(* Logix 5000 project; controller Project1Template vendor 1 type 14 code 151 rev 33.12; software revision 33.01 *)

TASK MainTask (continuous, watchdog 500 ms) : MainProgram

MODULES
   Local : vendor 1 type 14 code 151 (Compact 0, rev 33.12)
      Discrete_IO : Embedded (Compact 1, rev 3.1, Output RPI 20 ms)
      Analog_IO : Embedded (Compact 2, rev 1.1, Output RPI 80 ms)
      Counters : Embedded (Compact 3, rev 1.1, Output RPI 20 ms)
END_MODULES

TYPE Part_Type :
STRUCT
   Part_Name : STRING;
   Part_Number : INT;
   F1_HL : REAL;
   F1_LL : REAL;
   F2_HL : REAL;
   F2_LL : REAL;
   F3_HL : REAL;
   F3_LL : REAL;
   F4_HL : REAL;
   F4_LL : REAL;
   Active : BOOL;
   F1_Count : COUNTER;
   F2_Count : COUNTER;
   F3_Count : COUNTER;
   F4_Count : COUNTER;
END_STRUCT
END_TYPE

TYPE SHIFT_DATA :
STRUCT
   COMPLETED : DINT;
   PASSED : DINT;
   FAILED : DINT;
   EFFICIENT : REAL;
END_STRUCT
END_TYPE

ADD_ON_INSTRUCTION AOI_SIM_2PosCyl_ExtRet   (* revision 1.0 *)
VAR_OUTPUT
   Animation : DINT; {visible}
END_VAR
VAR_INPUT
   TravelTime : DINT; {required}
   Extend_Output : BOOL; {required}
   Retract_Output : BOOL; {required}
END_VAR
VAR_OUTPUT
   Extend_Sensor : BOOL; {access Read Only, required}
   Retract_Sensor : BOOL; {access Read Only, required}
END_VAR
VAR_INPUT
   MCR : BOOL; {required}
   SingleSolenoidExtend : BOOL; {required}
   SingleSolenoidRetract : BOOL; {required}
   Retract_ValvePB : BOOL;
   Extend_ValvePB : BOOL;
END_VAR
VAR
   Extend_ScanCount : DINT;
   Retract_ScanCount : DINT; {access None}
   Extend_Timer : TIMER := (PRE := 500); {access None}
   Retract_Timer : TIMER := (PRE := 500); {access None}
   Retracted : BOOL; {access None}
   Extended : BOOL; {access None}
   Retract : BOOL; {access None}
   Extend : BOOL; {access None}
END_VAR

ROUTINE Logic   (* ladder *)
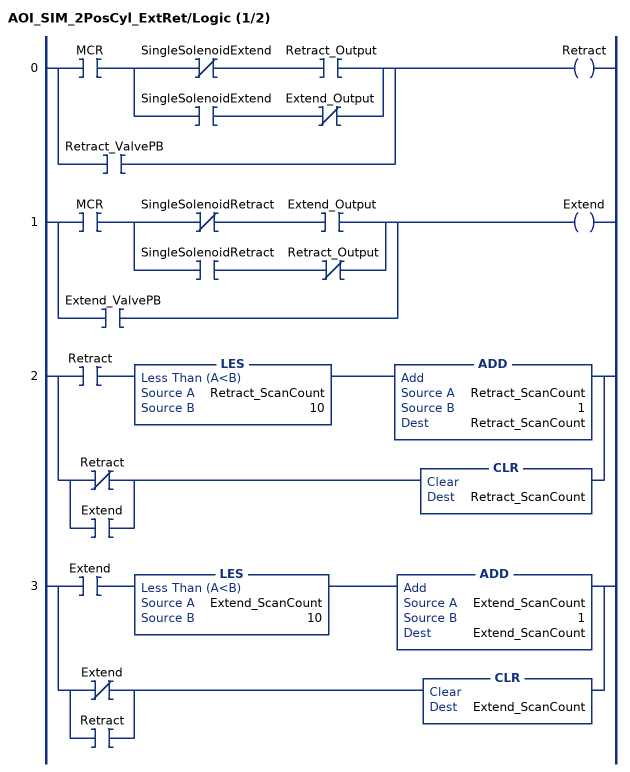
   0: [XIC(MCR) [XIO(SingleSolenoidExtend) XIC(Retract_Output) ,XIC(SingleSolenoidExtend) XIO(Extend_Output) ] ,XIC(Retract_ValvePB) ]OTE(Retract);
   1: [XIC(MCR) [XIO(SingleSolenoidRetract) XIC(Extend_Output) ,XIC(SingleSolenoidRetract) XIO(Retract_Output) ] ,XIC(Extend_ValvePB) ]OTE(Extend);
   2: [XIC(Retract) LES(Retract_ScanCount,10) ADD(Retract_ScanCount,1,Retract_ScanCount) ,[XIO(Retract) ,XIC(Extend) ] CLR(Retract_ScanCount) ];
   3: [XIC(Extend) LES(Extend_ScanCount,10) ADD(Extend_ScanCount,1,Extend_ScanCount) ,[XIO(Extend) ,XIC(Retract) ] CLR(Extend_ScanCount) ];
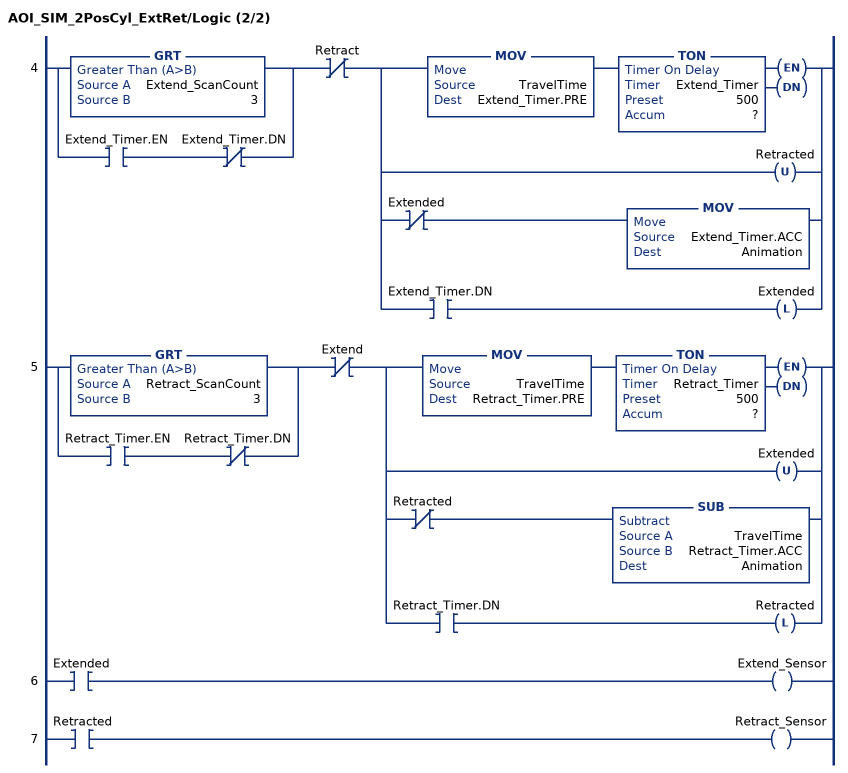
   4: [GRT(Extend_ScanCount,3) ,XIC(Extend_Timer.EN) XIO(Extend_Timer.DN) ]XIO(Retract)[MOV(TravelTime,Extend_Timer.PRE) TON(Extend_Timer,?,?) ,OTU(Retracted) ,XIO(Extended) MOV(Extend_Timer.ACC,Animation) ,XIC(Extend_Timer.DN) OTL(Extended) ];
   5: [GRT(Retract_ScanCount,3) ,XIC(Retract_Timer.EN) XIO(Retract_Timer.DN) ]XIO(Extend)[MOV(TravelTime,Retract_Timer.PRE) TON(Retract_Timer,?,?) ,OTU(Extended) ,XIO(Retracted) SUB(TravelTime,Retract_Timer.ACC,Animation) ,XIC(Retract_Timer.DN) OTL(Retracted) ];
   6: XIC(Extended)OTE(Extend_Sensor);
   7: XIC(Retracted)OTE(Retract_Sensor);
END_ROUTINE
END_ADD_ON_INSTRUCTION

ADD_ON_INSTRUCTION AOI_SIM_RandomDelay   (* revision 1.0 *)
VAR_INPUT
   Activate : BOOL; {access None}
   Target : DINT; {access None, required}
   Tolerance : DINT; {access None, required}
   PulseOutputTime : DINT; {access None, required}
END_VAR
VAR_OUTPUT
   DN : BOOL; {access Read Only, required}
END_VAR
VAR_INPUT
   DeActivate : BOOL; {access None}
END_VAR
VAR_OUTPUT
   TimingFirstHalf : BOOL; {access Read Only}
   TimingLastHalf : BOOL; {access Read Only}
   AccumlatedTime : DINT; {access Read Only}
   TT : BOOL; {access Read Only}
END_VAR
VAR
   StartTimerPulse : BOOL; {access None}
   StartTimerONS : BOOL; {access None}
   RandomIntermediate : DINT; {access None}
   RandomNumber : DINT; {access None}
   RandomPresetTime : DINT; {access None}
   RandomTimer : TIMER; {access None}
   PulseOutput : TIMER; {access None}
   Time50Percent : DINT; {access None}
END_VAR

ROUTINE Logic   (* ladder *)
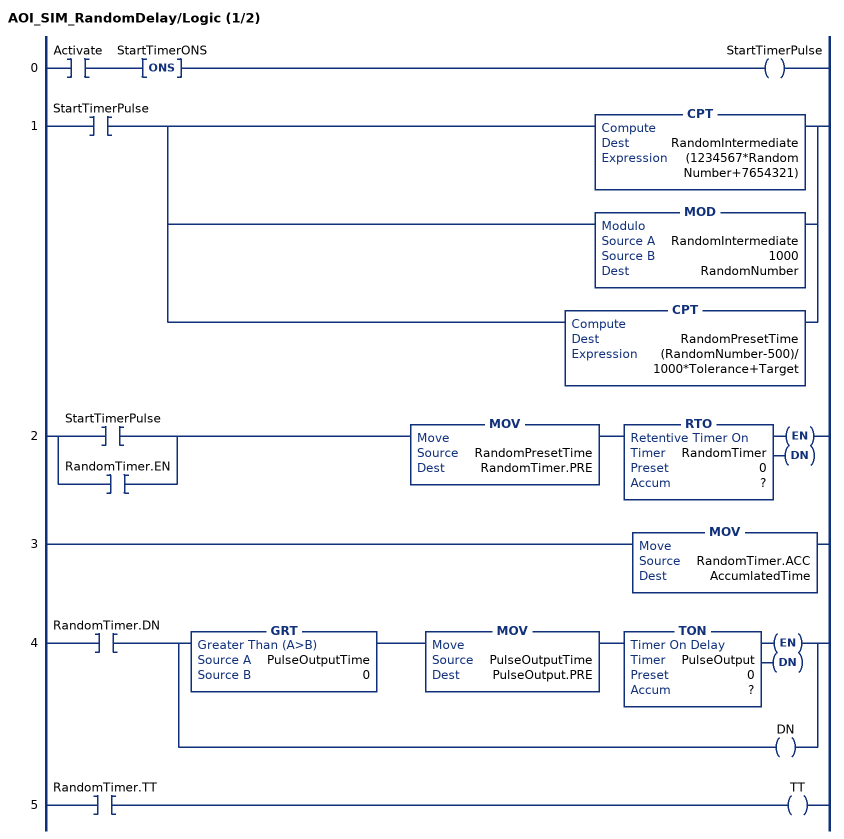
   0: XIC(Activate)ONS(StartTimerONS)OTE(StartTimerPulse);
   1: XIC(StartTimerPulse)[CPT(RandomIntermediate,(1234567*RandomNumber+7654321)) ,MOD(RandomIntermediate,1000,RandomNumber) ,CPT(RandomPresetTime,(RandomNumber-500)/1000*Tolerance+Target) ];
   2: [XIC(StartTimerPulse) ,XIC(RandomTimer.EN) ]MOV(RandomPresetTime,RandomTimer.PRE)RTO(RandomTimer,?,?);
   3: MOV(RandomTimer.ACC,AccumlatedTime);
   4: XIC(RandomTimer.DN)[GRT(PulseOutputTime,0) MOV(PulseOutputTime,PulseOutput.PRE) TON(PulseOutput,?,?) ,OTE(DN) ];
   5: XIC(RandomTimer.TT)OTE(TT);
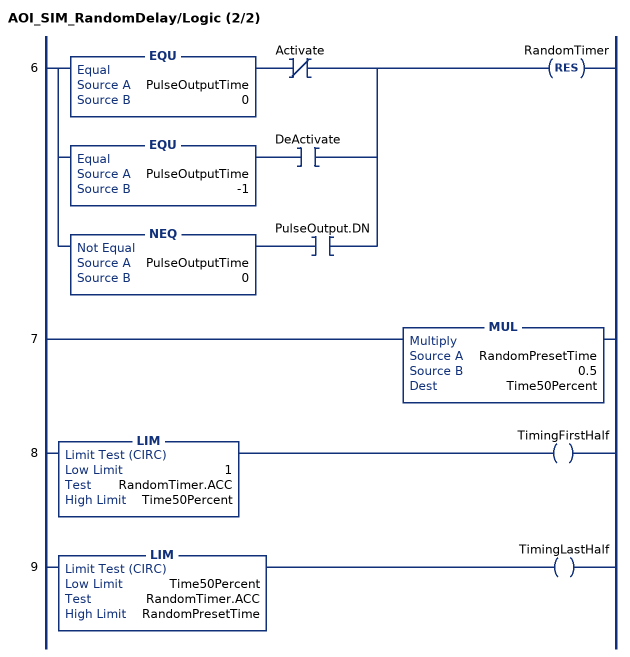
   6: [EQU(PulseOutputTime,0) XIO(Activate) ,EQU(PulseOutputTime,-1) XIC(DeActivate) ,NEQ(PulseOutputTime,0) XIC(PulseOutput.DN) ]RES(RandomTimer);
   7: MUL(RandomPresetTime,0.5,Time50Percent);
   8: LIM(1,RandomTimer.ACC,Time50Percent)OTE(TimingFirstHalf);
   9: LIM(Time50Percent,RandomTimer.ACC,RandomPresetTime)OTE(TimingLastHalf);
END_ROUTINE
END_ADD_ON_INSTRUCTION

ADD_ON_INSTRUCTION AOI_SIMAnalogSensor   (* revision 1.0 *)
VAR_IN_OUT
   Sensor : REAL; {required}
END_VAR
VAR_INPUT
   RampUpTime : DINT; {required}
   RampDwnTime : DINT; {required}
   Min : REAL; {required}
   Max : REAL; {required}
   Target : REAL; {required}
   Tolerance : REAL; {required}
   Fluctuation : REAL; {access None, required}
   Activate : BOOL; {access None}
END_VAR
VAR
   RampUpTimer : TIMER; {access None}
   RampDwnTimer : TIMER; {access None}
   FluctuateTimer : TIMER; {access None}
   FluctuateONS : BOOL; {access None}
   CurrentValue : REAL; {access Read Only}
   RampDwnTriggerONS : BOOL; {access Read Only}
   RampDwnTriggerPulse : BOOL; {access Read Only}
   RampUpTriggerONS : BOOL; {access Read Only}
   RampUpTriggerPulse : BOOL; {access Read Only}
   RandomNumber : DINT; {access Read Only}
   RandomTarget : REAL; {access Read Only}
   RandomIntermediate : DINT; {access Read Only}
   ScaledRampDwnTime : REAL; {access Read Only}
   ScaledRampUpTime : REAL; {access Read Only}
   Fluctuate : BOOL; {access None}
END_VAR

ROUTINE Logic   (* ladder *)
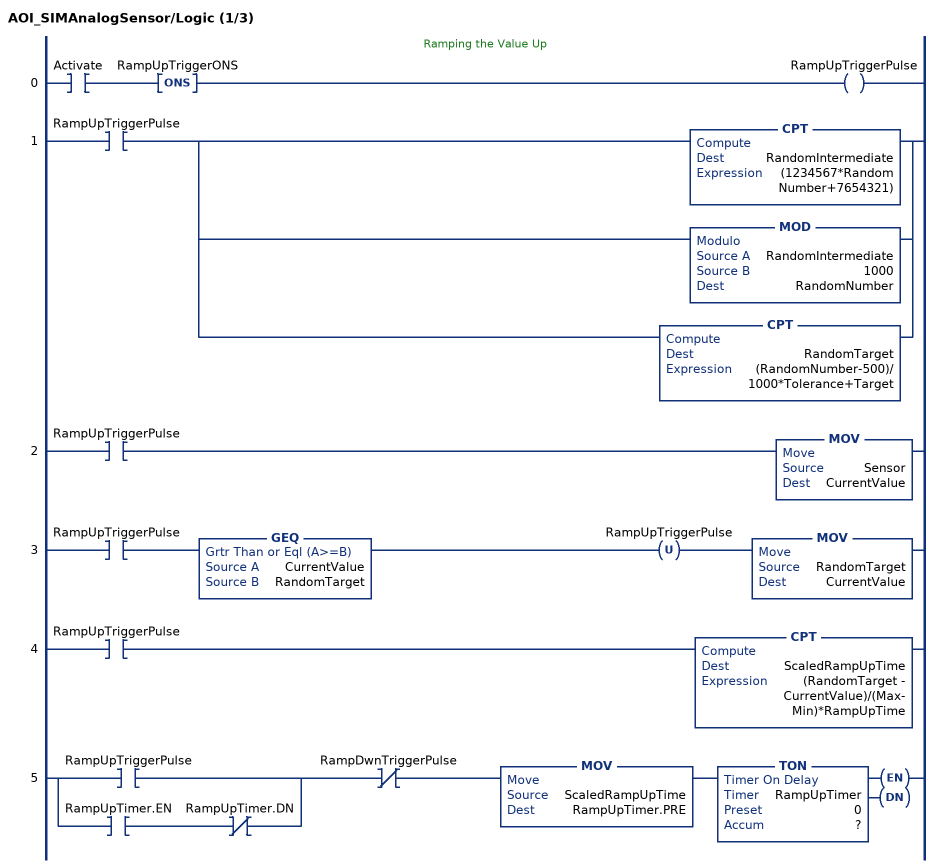
   // Ramping the Value Up
   0: XIC(Activate)ONS(RampUpTriggerONS)OTE(RampUpTriggerPulse);
   1: XIC(RampUpTriggerPulse)[CPT(RandomIntermediate,(1234567*RandomNumber+7654321)) ,MOD(RandomIntermediate,1000,RandomNumber) ,CPT(RandomTarget,(RandomNumber-500)/1000*Tolerance+Target) ];
   2: XIC(RampUpTriggerPulse)MOV(Sensor,CurrentValue);
   3: XIC(RampUpTriggerPulse)GEQ(CurrentValue,RandomTarget)OTU(RampUpTriggerPulse)MOV(RandomTarget,CurrentValue);
   4: XIC(RampUpTriggerPulse)CPT(ScaledRampUpTime,(RandomTarget - CurrentValue)/(Max-Min)*RampUpTime);
   5: [XIC(RampUpTriggerPulse) ,XIC(RampUpTimer.EN) XIO(RampUpTimer.DN) ]XIO(RampDwnTriggerPulse)MOV(ScaledRampUpTime,RampUpTimer.PRE)TON(RampUpTimer,?,?);
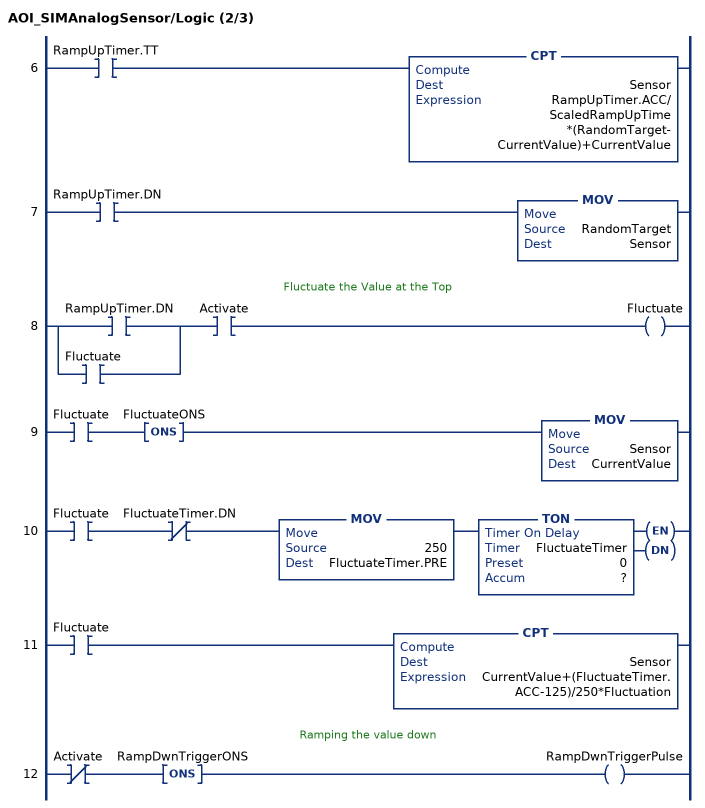
   6: XIC(RampUpTimer.TT)CPT(Sensor,RampUpTimer.ACC/ScaledRampUpTime *(RandomTarget-CurrentValue)+CurrentValue);
   7: XIC(RampUpTimer.DN)MOV(RandomTarget,Sensor);
   // Fluctuate the Value at the Top
   8: [XIC(RampUpTimer.DN) ,XIC(Fluctuate) ]XIC(Activate)OTE(Fluctuate);
   9: XIC(Fluctuate)ONS(FluctuateONS)MOV(Sensor,CurrentValue);
   10: XIC(Fluctuate)XIO(FluctuateTimer.DN)MOV(250,FluctuateTimer.PRE)TON(FluctuateTimer,?,?);
   11: XIC(Fluctuate)CPT(Sensor,CurrentValue+(FluctuateTimer.ACC-125)/250*Fluctuation);
   // Ramping the value down
   12: XIO(Activate)ONS(RampDwnTriggerONS)OTE(RampDwnTriggerPulse);
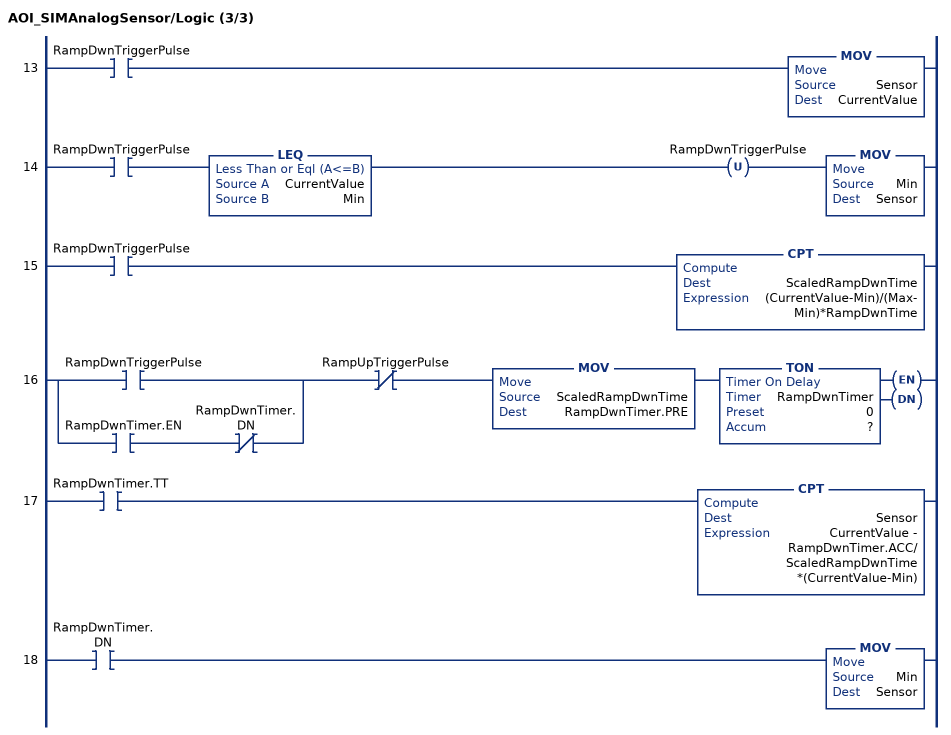
   13: XIC(RampDwnTriggerPulse)MOV(Sensor,CurrentValue);
   14: XIC(RampDwnTriggerPulse)LEQ(CurrentValue,Min)OTU(RampDwnTriggerPulse)MOV(Min,Sensor);
   15: XIC(RampDwnTriggerPulse)CPT(ScaledRampDwnTime,(CurrentValue-Min)/(Max-Min)*RampDwnTime);
   16: [XIC(RampDwnTriggerPulse) ,XIC(RampDwnTimer.EN) XIO(RampDwnTimer.DN) ]XIO(RampUpTriggerPulse)MOV(ScaledRampDwnTime,RampDwnTimer.PRE)TON(RampDwnTimer,?,?);
   17: XIC(RampDwnTimer.TT)CPT(Sensor,CurrentValue - RampDwnTimer.ACC/ScaledRampDwnTime *(CurrentValue-Min));
   18: XIC(RampDwnTimer.DN)MOV(Min,Sensor);
END_ROUTINE
END_ADD_ON_INSTRUCTION

VAR_GLOBAL   (* controller tags *)
   A_EXT_TMR : TIMER := (PRE := 10000);
   A_RET_TMR : TIMER := (PRE := 10000);
   ADD12 : DINT := 4;
   ADD123 : DINT := 6;
   ADD123FAIL : DINT := 3;
   ADD123PASS : DINT := 3;
   ADD12FAIL : DINT := 2;
   ADD12PASS : DINT := 2;
   ALLFAILONES : BOOL;
   AVERAGE1 : CONTROL := (LEN := 50);
   AVERAGECNTRL : CONTROL := (LEN := 50);
   B_EXT_TMR : TIMER := (PRE := 10000);
   B_RET_TMR : TIMER := (PRE := 10000);
   Batch_Count : INT;
   C_EXT_TMR : TIMER := (PRE := 10000);
   C_RET_TMR : TIMER := (PRE := 10000);
   CHANGED : BOOL;
   CHANGEONS : BOOL;
   Current_Part : Part_Type;
   Current_Part_Count : INT;
   Current_Part_Name : STRING;
   Current_Part_Number : INT;
   CURRENT_SHIFT : SHIFT_DATA := (COMPLETED := 8, PASSED := 5, FAILED := 3, EFFICIENT := 62.5);
   CURRENT_TOTAL_COUNT : DINT;
   DATASHIFT : BOOL;
   EFFICIENCY : REAL;
   END_SHIFT_PB : BOOL;
   EStop : BOOL;
   EXTRA_TIME : TIMER := (PRE := 120000);
   F1_AVERAGE : REAL := 44.42104;
   F1_Count : COUNTER := (ACC := 2, DN := 1);
   F1_CT_AVERAGE : REAL := 1000.2;
   F1_CT_History : REAL[5] := ([0] := 2501.0, [2] := 2500.0);
   F1_Current_Part_Count : DINT;
   F1_FAIL : COUNTER := (ACC := 1, DN := 1);
   F1_PASS : COUNTER := (ACC := 1, DN := 1);
   F1_TEMP_TORQUE : DINT[50];
   F1_TORQUE : REAL[50];
   F1_Torque_History : REAL[5] := ([0] := 75.627594, [1] := 73.2388, [2] := 73.2388);
   F2_Count : COUNTER := (ACC := 2, DN := 1);
   F2_CT_AVERAGE : REAL := 3399.4;
   F2_CT_History : REAL[5] := ([0] := 3499.0, [2] := 13498.0);
   F2_Current_Part_Count : DINT;
   F2_FAIL : COUNTER := (ACC := 1, DN := 1);
   F2_PASS : COUNTER := (ACC := 1, DN := 1);
   F2_Torque_History : REAL[5] := ([0] := 74.103195, [1] := 73.3064, [2] := 73.3064);
   F3_Count : COUNTER := (ACC := 2, DN := 1);
   F3_CT_AVERAGE : REAL := 3799.8;
   F3_CT_History : REAL[5] := ([0] := 4499.0, [2] := 14500.0);
   F3_Current_Part_Count : DINT;
   F3_FAIL : COUNTER := (ACC := 1, DN := 1);
   F3_PASS : COUNTER := (ACC := 1, DN := 1);
   F3_Torque_History : REAL[5] := ([0] := 76.578, [1] := 72.995605, [2] := 72.995605);
   F4_Count : COUNTER := (ACC := 2, DN := 1);
   F4_CT_AVERAGE : REAL := 3499.6;
   F4_CT_History : REAL[5] := ([0] := 3749.0, [2] := 13749.0);
   F4_Current_Part_Count : DINT;
   F4_FAIL : COUNTER := (DN := 1);
   F4_PASS : COUNTER := (ACC := 2, DN := 1);
   F4_Torque_History : REAL[5] := ([0] := 78.5, [1] := 77.1048, [2] := 77.1048);
   F_ALL_CTR : COUNTER := (ACC := 1);
   FAILONS1 : BOOL;
   FAILONS2 : BOOL;
   FAILONS3 : BOOL;
   FAILONS4 : BOOL;
   FASTEN_AllComplete : BOOL;
   FASTEN_AllTorquesFail : BOOL;
   FASTEN_AllTorquesPass : BOOL;
   FASTEN_F1Complete : BOOL;
   FASTEN_F1Complete_ONS : BOOL;
   FASTEN_F1Torque : REAL;
   FASTEN_F1TorqueFail : BOOL;
   FASTEN_F1TorquePass : BOOL;
   FASTEN_F2Complete : BOOL;
   FASTEN_F2Complete_ONS : BOOL;
   FASTEN_F2Torque : REAL;
   FASTEN_F2TorqueFail : BOOL;
   FASTEN_F2TorquePass : BOOL;
   FASTEN_F3Complete : BOOL;
   FASTEN_F3Complete_ONS : BOOL;
   FASTEN_F3Torque : REAL;
   FASTEN_F3TorqueFail : BOOL;
   FASTEN_F3TorquePass : BOOL;
   FASTEN_F4Complete : BOOL;
   FASTEN_F4Complete_ONS : BOOL;
   FASTEN_F4Torque : REAL;
   FASTEN_F4TorqueFail : BOOL;
   FASTEN_F4TorquePass : BOOL;
   FASTEN_TorqueFeedback : REAL := 20.050001;
   FAULTRESET_PB : BOOL;
   FAULTS : DINT;
   FAULTSIND : BOOL;
   FIX_EXT_TMR : TIMER := (PRE := 10000);
   FIX_RET_TMR : TIMER := (PRE := 10000);
   FIXTURE_AllPartsPresent : BOOL := 1;
   FIXTURE_AtHomePos : BOOL := 1;
   FIXTURE_Empty : BOOL;
   FIXTURE_PartsSecured : BOOL;
   FIXTURE_PartsSecuredTmr : TIMER := (PRE := 500);
   FromHMI_ExtClampA_PB : BOOL;
   FromHMI_ExtClampB_PB : BOOL;
   FromHMI_ExtClampC_PB : BOOL;
   FromHMI_ExtFixture_PB : BOOL;
   FromHMI_F1LowLim : REAL := 50.0;
   FromHMI_F1UppLim : REAL := 95.0;
   FromHMI_F2LowLim : REAL := 65.0;
   FromHMI_F2UppLim : REAL := 85.0;
   FromHMI_F3LowLim : REAL := 60.0;
   FromHMI_F3UppLim : REAL := 85.0;
   FromHMI_F4LowLim : REAL := 66.0;
   FromHMI_F4UppLim : REAL := 95.0;
   FromHMI_RetClampA_PB : BOOL;
   FromHMI_RetClampB_PB : BOOL;
   FromHMI_RetClampC_PB : BOOL;
   FromHMI_RetFixture_PB : BOOL;
   FROMHMI_SCREEN : DINT;
   FromHMI_StartPB : BOOL;
   FromHMI_StopPB : BOOL;
   FromRbt_ClearOfFixture : BOOL := 1;
   FromRbt_Fasten1Complete : BOOL;
   FromRbt_Fasten2Complete : BOOL;
   FromRbt_Fasten3Complete : BOOL;
   FromRbt_Fasten4Complete : BOOL;
   HomePB : BOOL;
   Honda : STRING := 'Honda';
   I1 : INT := 20318;
        .10   // Part Present C Sensor
        .11   // Part Present D Sensor
        .14   // Light Curtain Safety Circuit
        .0   // Fixture at Robot Limit Switch
        .1   // Fixture at Operator Limit Switch
        .2   // Clamp A Retracted Limit Switch
        .3   // Clamp B Retracted Limit Switch
        .4   // Clamp C Retracted Limit Switch
        .8   // Part Present A Sensor
        .9   // Part Present B Sensor
   I2_CHA : REAL := 4.01;   // Torque Sensor Input
   Lexus : STRING := 'Lexus';
   Load_PB : BOOL;
   O3 : INT;
        .1   // Fixture Retract to Operator
        .3   // Clamp B Extend Solenoid
        .0   // Fixture Extend to Robot
        .2   // Clamp A Extend Solenoid
        .4   // Clamp C Extend Solenoid
   ONEHR : BOOL;
   ONS1 : BOOL;
   ONS2 : BOOL;
   ONS3 : BOOL;
   ONS4 : BOOL;
   P1_ADD12 : DINT;
   P1_ADD123 : DINT;
   P2_ADD12 : DINT;
   P2_ADD123 : DINT;
   P3_ADD12 : DINT;
   P3_ADD123 : DINT;
   PART1 : Part_Type := (Part_Name := 'toyota', Part_Number := 1, F1_HL := 95.0, F1_LL := 75.0, F2_HL := 85.0, F2_LL := 75.0, F3_HL := 85.0, F3_LL := 75.0, F4_HL := 95.0, F4_LL := 75.0, F1_Count.DN := 1, F2_Count.DN := 1, F3_Count.DN := 1, F4_Count.DN := 1);
   PART2 : Part_Type := (F1_Count.DN := 1, F2_Count.DN := 1, F3_Count.DN := 1, F4_Count.DN := 1);
   PART3 : Part_Type := (Part_Name := 'Honda', Part_Number := 3, F1_HL := 95.0, F1_LL := 50.0, F2_HL := 85.0, F2_LL := 65.0, F3_HL := 85.0, F3_LL := 60.0, F4_HL := 95.0, F4_LL := 66.0, F1_Count.DN := 1, F2_Count.DN := 1, F3_Count.DN := 1, F4_Count.DN := 1);
   Part_Name : STRING;
   Part_Number : DINT := 3;
   Requested_Part_Number : INT;
   RESET_STATS : BOOL;
   S1ON : BOOL;
   SCREENREQTMR : TIMER := (PRE := 1000);
   SHIFT1ONS : BOOL;
   SHIFT_CHANGE : BOOL;
   SHIFT_TIMER : TIMER := (PRE := 120000);
   SHIFTHISTORY : SHIFT_DATA[5];
   SHIFTONS : BOOL;
   STARTONS : BOOL;
   SYS_AutoModeActive : BOOL := 1;
   SYS_CycleActive : BOOL;
   SYS_ManualModeActive : BOOL;
   SYS_StartPBPulseTmr : TIMER := (PRE := 200);
   T1AVG : DINT;
   THREEHR : BOOL;
   TIME : REAL;
   TOHMI_CHANGEVALVE : BOOL;
   TOHMI_CHANGEWARNING : BOOL;
   TOHMI_SCREENREQ : DINT;
   ToRbt_Fasten1Start : BOOL;
   ToRbt_Fasten2Start : BOOL;
   ToRbt_Fasten3Start : BOOL;
   ToRbt_Fasten4Start : BOOL;
   Total_Parts : INT;
   TOTAL_PARTS_COMPLETE : DINT;
   TOTAL_PARTS_FAIL : DINT;
   TOTAL_PARTS_PASS : DINT;
   Toyota : STRING := 'toyota';
   TWOHR : BOOL;
   VALVECTR : COUNTER := (ACC := 10, DN := 1);
   VALVEONS : BOOL;
   VALVEWARNING : DINT;
END_VAR

PROGRAM MainProgram   (* main routine MainRoutine *)
VAR
   Cycle_Time_Calc : TIMER := (PRE := 9999999);
   F1_CycleTime : REAL := 2501.0;
   F2_AVERAGE : REAL := 44.143196;
   F2_CycleTime : REAL := 3499.0;
   F2_TMR : TIMER := (PRE := 9999999);
   F3_AVERAGE : REAL := 44.513844;
   F3_CycleTime : REAL := 4499.0;
   F3_TMR : TIMER := (PRE := 9999999);
   F4_AVERAGE : REAL := 46.54192;
   F4_CycleTime : REAL := 3749.0;
   F4_TMR : TIMER := (PRE := 9999999);
   ONS_CTH : BOOL;
   ONS_F1_CT : BOOL;
   ONS_TH : BOOL;
   SIM_ClampA : AOI_SIM_2PosCyl_ExtRet := (TravelTime := 1000, Retract_Sensor := 1, MCR := 1, SingleSolenoidExtend := 1);
   SIM_ClampB : AOI_SIM_2PosCyl_ExtRet := (TravelTime := 1250, Retract_Sensor := 1, MCR := 1, SingleSolenoidExtend := 1);
   SIM_ClampC : AOI_SIM_2PosCyl_ExtRet := (TravelTime := 1250, Retract_Sensor := 1, MCR := 1, SingleSolenoidExtend := 1);
   SIM_EmptyFixture : TIMER := (PRE := 15000);
   SIM_Fasten1 : AOI_SIM_RandomDelay := (Target := 2500, Tolerance := 750);
   SIM_Fasten2 : AOI_SIM_RandomDelay := (Target := 3500, Tolerance := 450);
   SIM_Fasten3 : AOI_SIM_RandomDelay := (Target := 4500, Tolerance := 250);
   SIM_Fasten4 : AOI_SIM_RandomDelay := (Target := 3750, Tolerance := 500);
   SIM_Fixture : AOI_SIM_2PosCyl_ExtRet := (TravelTime := 2000, Retract_Sensor := 1, MCR := 1);
   SIM_LightCurtainPartPlace : AOI_SIM_RandomDelay := (Target := 6000, Tolerance := 1500, PulseOutputTime := 50);
   SIM_LightCurtainPartRem : AOI_SIM_RandomDelay := (Target := 5000, Tolerance := 1000, PulseOutputTime := 50);
   SIM_NOP : BOOL;
   SIM_Oneshots : DINT := 1;
   SIM_OperatorWorking : AOI_SIM_RandomDelay := (Target := 4000, Tolerance := 2000, PulseOutputTime := 50);
   SIM_PP_OFF : AOI_SIM_RandomDelay := (Target := 2500, Tolerance := 1000, PulseOutputTime := 50);
   SIM_PPA_ON : AOI_SIM_RandomDelay := (Target := 1500, Tolerance := 500, PulseOutputTime := 50);
   SIM_PPB_ON : AOI_SIM_RandomDelay := (Target := 2000, Tolerance := 1000, PulseOutputTime := 50);
   SIM_PPC_ON : AOI_SIM_RandomDelay := (Target := 2500, Tolerance := 1000, PulseOutputTime := 50);
   SIM_PPD_ON : AOI_SIM_RandomDelay := (Target := 3000, Tolerance := 500, PulseOutputTime := 50);
   SIM_RobotClear : AOI_SIM_RandomDelay := (Target := 1200, Tolerance := 250, PulseOutputTime := 50);
   SIM_Torque : AOI_SIMAnalogSensor := (RampUpTime := 500, RampDwnTime := 50, Min := 4.01, Max := 19.99, Target := 15.0, Tolerance := 2.0, Fluctuation := 0.04);
END_VAR

ROUTINE EXTRAS   (* ladder *)
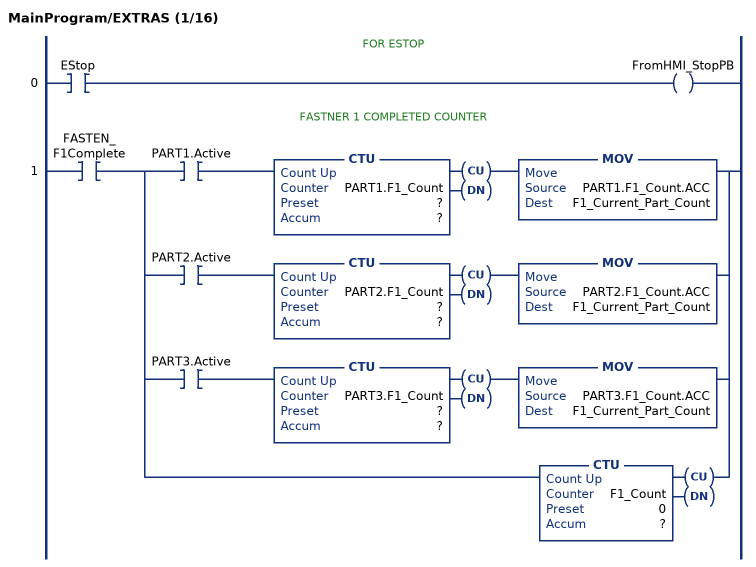
   // FOR ESTOP
   0: XIC(EStop)OTE(FromHMI_StopPB);
   // FASTNER 1 COMPLETED COUNTER
   1: XIC(FASTEN_F1Complete)[XIC(PART1.Active) CTU(PART1.F1_Count,?,?) MOV(PART1.F1_Count.ACC,F1_Current_Part_Count) ,XIC(PART2.Active) CTU(PART2.F1_Count,?,?) MOV(PART2.F1_Count.ACC,F1_Current_Part_Count) ,XIC(PART3.Active) CTU(PART3.F1_Count,?,?) MOV(PART3.F1_Count.ACC,F1_Current_Part_Count) ,CTU(F1_Count,?,?) ];
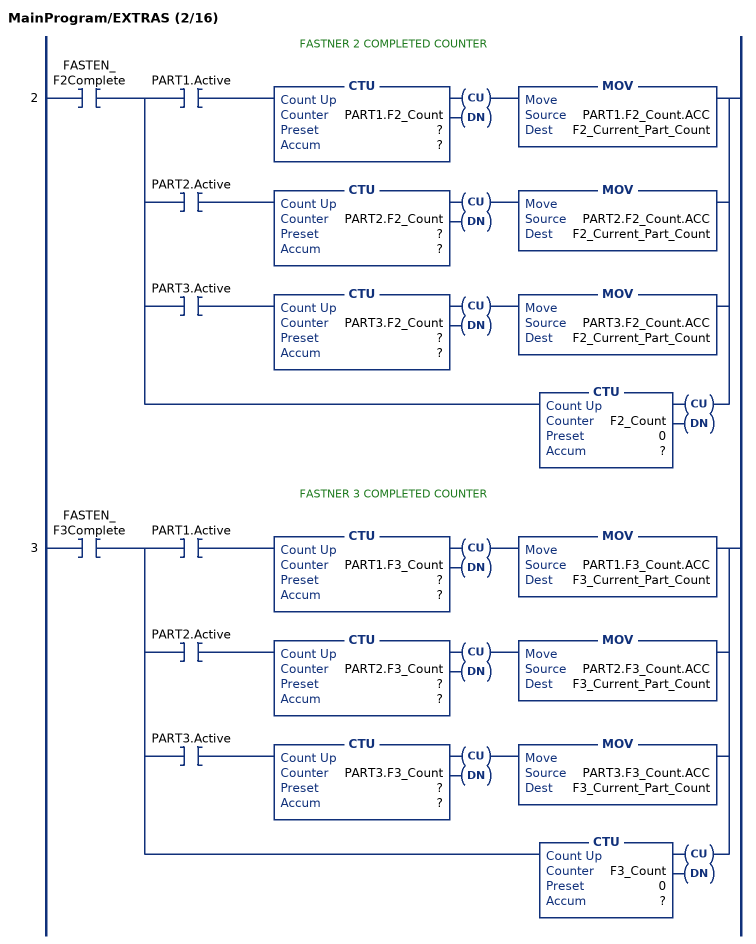
   // FASTNER 2 COMPLETED COUNTER
   2: XIC(FASTEN_F2Complete)[XIC(PART1.Active) CTU(PART1.F2_Count,?,?) MOV(PART1.F2_Count.ACC,F2_Current_Part_Count) ,XIC(PART2.Active) CTU(PART2.F2_Count,?,?) MOV(PART2.F2_Count.ACC,F2_Current_Part_Count) ,XIC(PART3.Active) CTU(PART3.F2_Count,?,?) MOV(PART3.F2_Count.ACC,F2_Current_Part_Count) ,CTU(F2_Count,?,?) ];
   // FASTNER 3 COMPLETED COUNTER
   3: XIC(FASTEN_F3Complete)[XIC(PART1.Active) CTU(PART1.F3_Count,?,?) MOV(PART1.F3_Count.ACC,F3_Current_Part_Count) ,XIC(PART2.Active) CTU(PART2.F3_Count,?,?) MOV(PART2.F3_Count.ACC,F3_Current_Part_Count) ,XIC(PART3.Active) CTU(PART3.F3_Count,?,?) MOV(PART3.F3_Count.ACC,F3_Current_Part_Count) ,CTU(F3_Count,?,?) ];
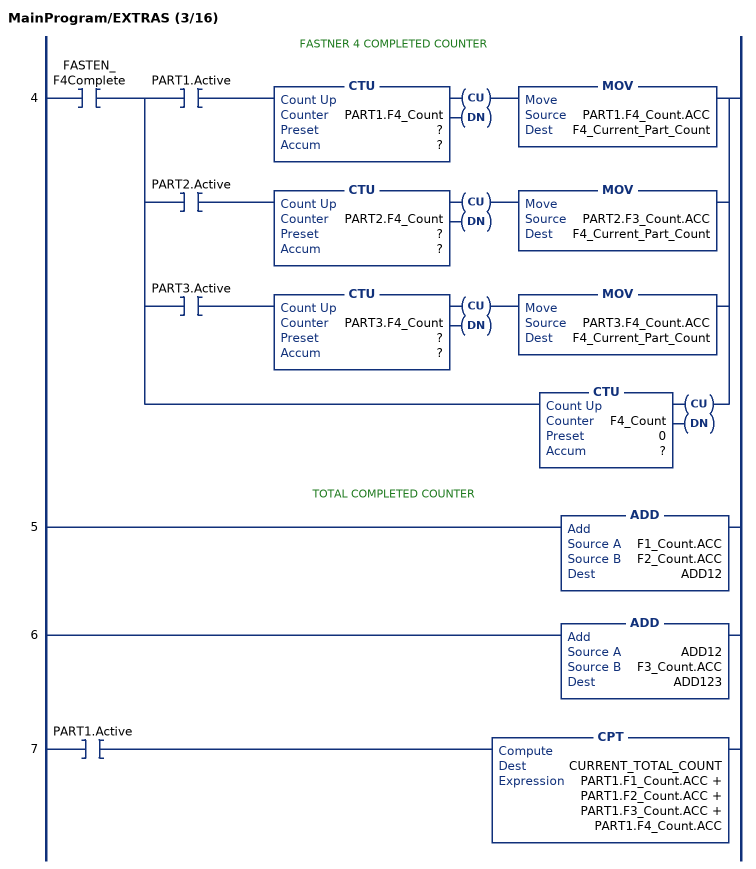
   // FASTNER 4 COMPLETED COUNTER
   4: XIC(FASTEN_F4Complete)[XIC(PART1.Active) CTU(PART1.F4_Count,?,?) MOV(PART1.F4_Count.ACC,F4_Current_Part_Count) ,XIC(PART2.Active) CTU(PART2.F4_Count,?,?) MOV(PART2.F3_Count.ACC,F4_Current_Part_Count) ,XIC(PART3.Active) CTU(PART3.F4_Count,?,?) MOV(PART3.F4_Count.ACC,F4_Current_Part_Count) ,CTU(F4_Count,?,?) ];
   // TOTAL COMPLETED COUNTER
   5: ADD(F1_Count.ACC,F2_Count.ACC,ADD12);
   6: ADD(ADD12,F3_Count.ACC,ADD123);
   7: XIC(PART1.Active)CPT(CURRENT_TOTAL_COUNT,PART1.F1_Count.ACC + PART1.F2_Count.ACC + PART1.F3_Count.ACC + PART1.F4_Count.ACC);
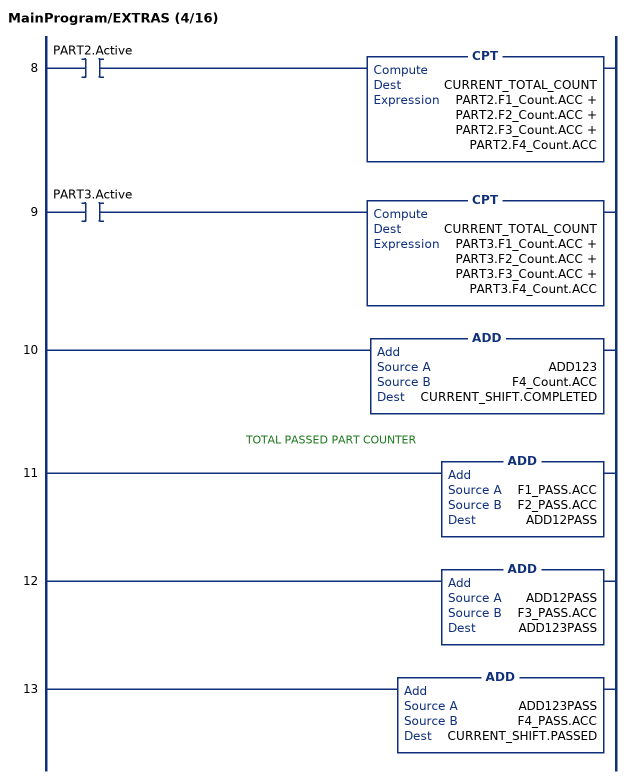
   8: XIC(PART2.Active)CPT(CURRENT_TOTAL_COUNT,PART2.F1_Count.ACC + PART2.F2_Count.ACC + PART2.F3_Count.ACC + PART2.F4_Count.ACC);
   9: XIC(PART3.Active)CPT(CURRENT_TOTAL_COUNT,PART3.F1_Count.ACC + PART3.F2_Count.ACC + PART3.F3_Count.ACC + PART3.F4_Count.ACC);
   10: ADD(ADD123,F4_Count.ACC,CURRENT_SHIFT.COMPLETED);
   // TOTAL PASSED PART COUNTER
   11: ADD(F1_PASS.ACC,F2_PASS.ACC,ADD12PASS);
   12: ADD(ADD12PASS,F3_PASS.ACC,ADD123PASS);
   13: ADD(ADD123PASS,F4_PASS.ACC,CURRENT_SHIFT.PASSED);
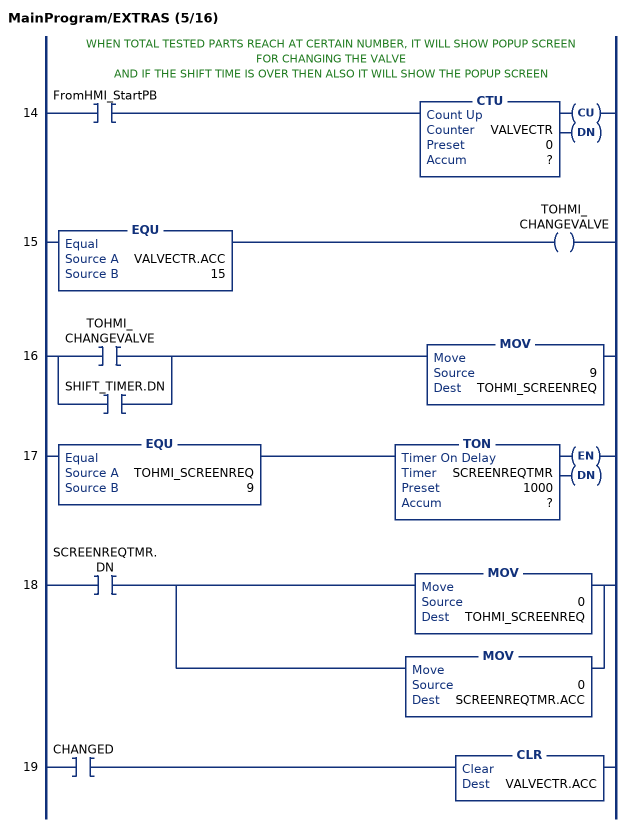
   // WHEN TOTAL TESTED PARTS REACH AT CERTAIN NUMBER, IT WILL SHOW POPUP SCREEN FOR CHANGING THE VALVE
   // AND IF THE SHIFT TIME IS OVER THEN ALSO IT WILL SHOW THE POPUP SCREEN
   14: XIC(FromHMI_StartPB)CTU(VALVECTR,?,?);
   15: EQU(VALVECTR.ACC,15)OTE(TOHMI_CHANGEVALVE);
   16: [XIC(TOHMI_CHANGEVALVE) ,XIC(SHIFT_TIMER.DN) ]MOV(9,TOHMI_SCREENREQ);
   17: EQU(TOHMI_SCREENREQ,9)TON(SCREENREQTMR,?,?);
   18: XIC(SCREENREQTMR.DN)[MOV(0,TOHMI_SCREENREQ) ,MOV(0,SCREENREQTMR.ACC) ];
   19: XIC(CHANGED)CLR(VALVECTR.ACC);
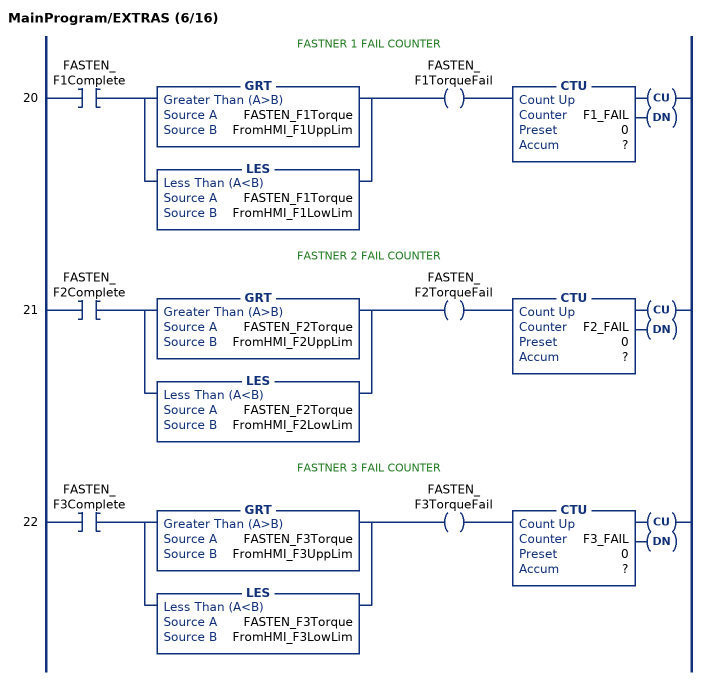
   // FASTNER 1 FAIL COUNTER
   20: XIC(FASTEN_F1Complete)[GRT(FASTEN_F1Torque,FromHMI_F1UppLim) ,LES(FASTEN_F1Torque,FromHMI_F1LowLim) ]OTE(FASTEN_F1TorqueFail)CTU(F1_FAIL,?,?);
   // FASTNER 2 FAIL COUNTER
   21: XIC(FASTEN_F2Complete)[GRT(FASTEN_F2Torque,FromHMI_F2UppLim) ,LES(FASTEN_F2Torque,FromHMI_F2LowLim) ]OTE(FASTEN_F2TorqueFail)CTU(F2_FAIL,?,?);
   // FASTNER 3 FAIL COUNTER
   22: XIC(FASTEN_F3Complete)[GRT(FASTEN_F3Torque,FromHMI_F3UppLim) ,LES(FASTEN_F3Torque,FromHMI_F3LowLim) ]OTE(FASTEN_F3TorqueFail)CTU(F3_FAIL,?,?);
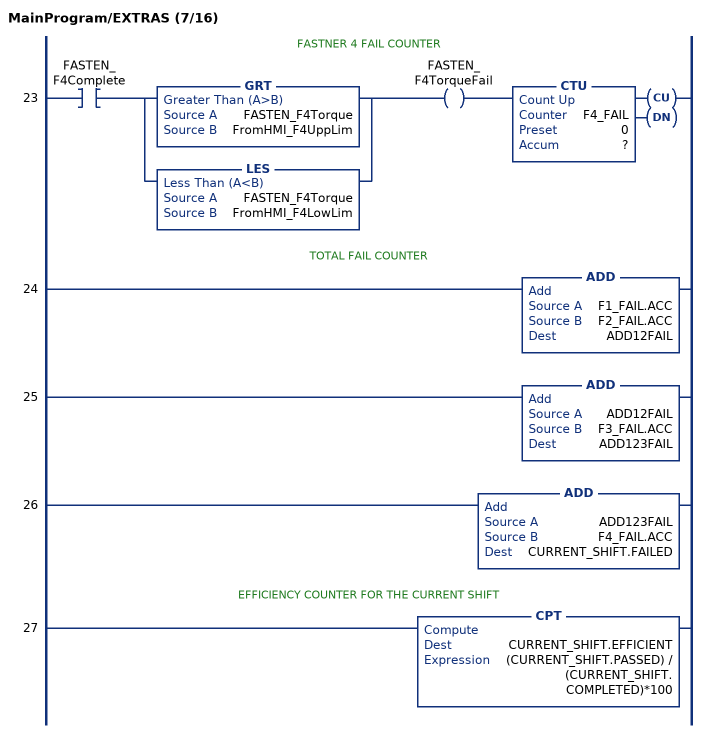
   // FASTNER 4 FAIL COUNTER
   23: XIC(FASTEN_F4Complete)[GRT(FASTEN_F4Torque,FromHMI_F4UppLim) ,LES(FASTEN_F4Torque,FromHMI_F4LowLim) ]OTE(FASTEN_F4TorqueFail)CTU(F4_FAIL,?,?);
   // TOTAL FAIL COUNTER
   24: ADD(F1_FAIL.ACC,F2_FAIL.ACC,ADD12FAIL);
   25: ADD(ADD12FAIL,F3_FAIL.ACC,ADD123FAIL);
   26: ADD(ADD123FAIL,F4_FAIL.ACC,CURRENT_SHIFT.FAILED);
   // EFFICIENCY COUNTER FOR THE CURRENT SHIFT
   27: CPT(CURRENT_SHIFT.EFFICIENT,(CURRENT_SHIFT.PASSED) / (CURRENT_SHIFT.COMPLETED)*100);
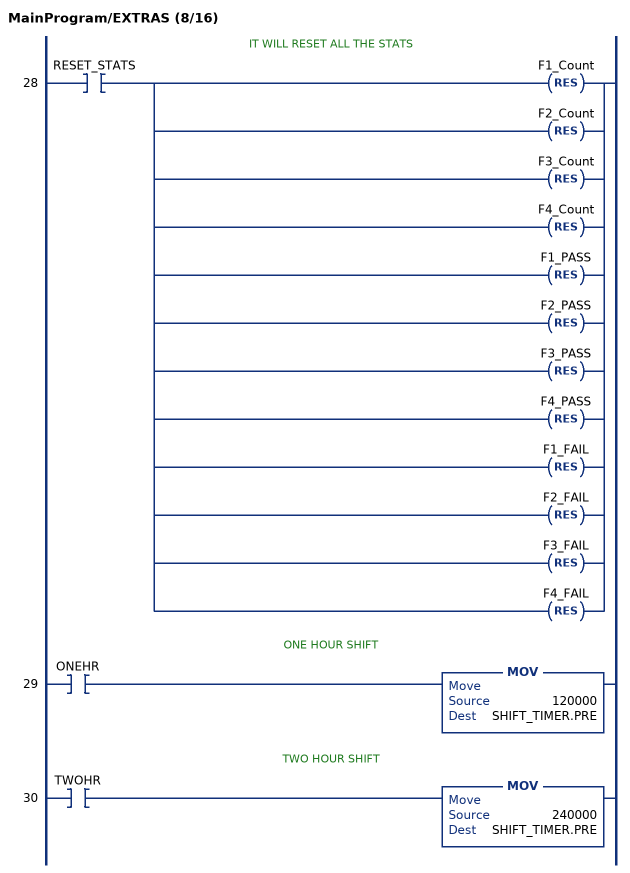
   // IT WILL RESET ALL THE STATS
   28: XIC(RESET_STATS)[RES(F1_Count) ,RES(F2_Count) ,RES(F3_Count) ,RES(F4_Count) ,RES(F1_PASS) ,RES(F2_PASS) ,RES(F3_PASS) ,RES(F4_PASS) ,RES(F1_FAIL) ,RES(F2_FAIL) ,RES(F3_FAIL) ,RES(F4_FAIL) ];
   // ONE HOUR SHIFT
   29: XIC(ONEHR)MOV(120000,SHIFT_TIMER.PRE);
   // TWO HOUR SHIFT
   30: XIC(TWOHR)MOV(240000,SHIFT_TIMER.PRE);
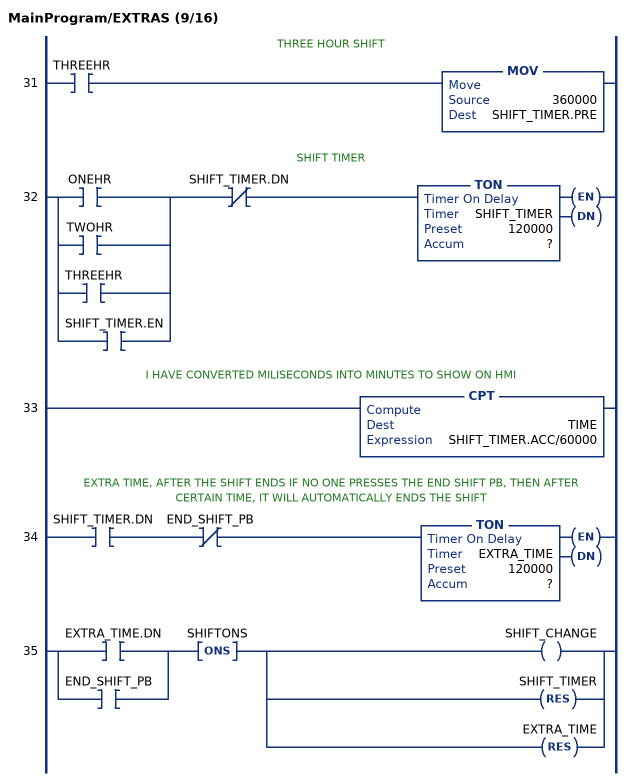
   // THREE HOUR SHIFT
   31: XIC(THREEHR)MOV(360000,SHIFT_TIMER.PRE);
   // SHIFT TIMER
   32: [[XIC(ONEHR) ,XIC(TWOHR) ,XIC(THREEHR) ] ,XIC(SHIFT_TIMER.EN) ]XIO(SHIFT_TIMER.DN)TON(SHIFT_TIMER,?,?);
   // I HAVE CONVERTED MILISECONDS INTO MINUTES TO SHOW ON HMI
   33: CPT(TIME,SHIFT_TIMER.ACC/60000);
   // EXTRA TIME, AFTER THE SHIFT ENDS IF NO ONE PRESSES THE END SHIFT PB, THEN AFTER CERTAIN TIME, IT WILL AUTOMATICALLY ENDS THE SHIFT
   34: XIC(SHIFT_TIMER.DN)XIO(END_SHIFT_PB)TON(EXTRA_TIME,?,?);
   35: [XIC(EXTRA_TIME.DN) ,XIC(END_SHIFT_PB) ]ONS(SHIFTONS)[OTE(SHIFT_CHANGE) ,RES(SHIFT_TIMER) ,RES(EXTRA_TIME) ];
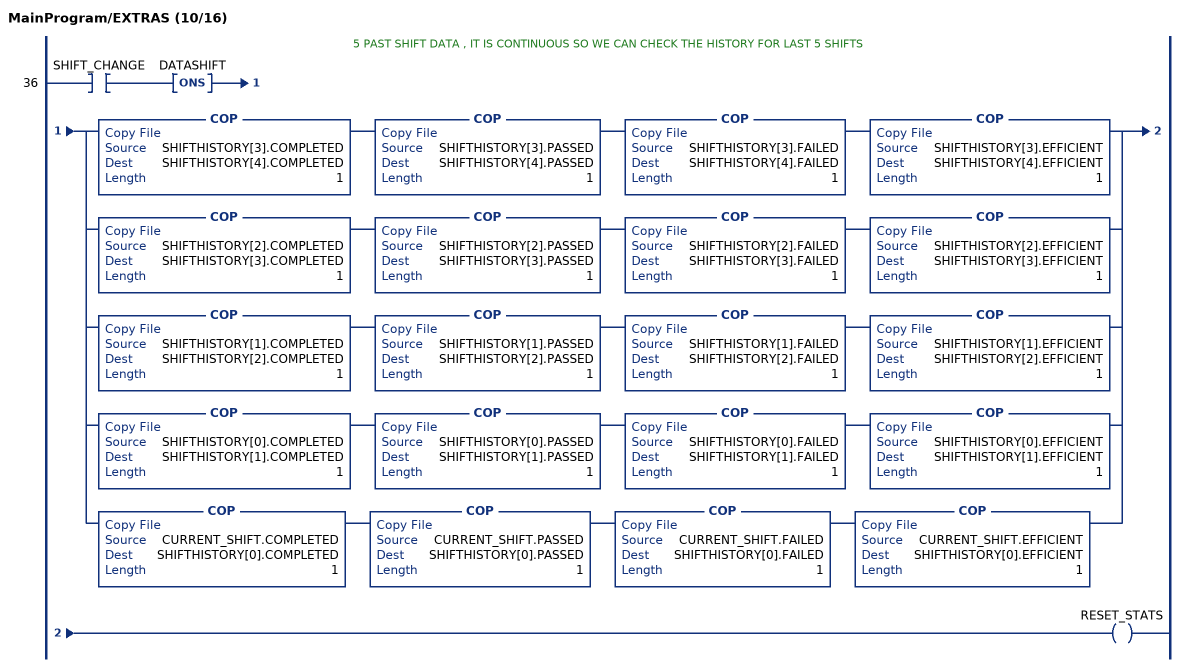
   // 5 PAST SHIFT DATA , IT IS CONTINUOUS SO WE CAN CHECK THE HISTORY FOR LAST 5 SHIFTS
   36: XIC(SHIFT_CHANGE)ONS(DATASHIFT)[COP(SHIFTHISTORY[3].COMPLETED,SHIFTHISTORY[4].COMPLETED,1) COP(SHIFTHISTORY[3].PASSED,SHIFTHISTORY[4].PASSED,1) COP(SHIFTHISTORY[3].FAILED,SHIFTHISTORY[4].FAILED,1) COP(SHIFTHISTORY[3].EFFICIENT,SHIFTHISTORY[4].EFFICIENT,1) ,COP(SHIFTHISTORY[2].COMPLETED,SHIFTHISTORY[3].COMPLETED,1) COP(SHIFTHISTORY[2].PASSED,SHIFTHISTORY[3].PASSED,1) COP(SHIFTHISTORY[2].FAILED,SHIFTHISTORY[3].FAILED,1) COP(SHIFTHISTORY[2].EFFICIENT,SHIFTHISTORY[3].EFFICIENT,1) ,COP(SHIFTHISTORY[1].COMPLETED,SHIFTHISTORY[2].COMPLETED,1) COP(SHIFTHISTORY[1].PASSED,SHIFTHISTORY[2].PASSED,1) COP(SHIFTHISTORY[1].FAILED,SHIFTHISTORY[2].FAILED,1) COP(SHIFTHISTORY[1].EFFICIENT,SHIFTHISTORY[2].EFFICIENT,1) ,COP(SHIFTHISTORY[0].COMPLETED,SHIFTHISTORY[1].COMPLETED,1) COP(SHIFTHISTORY[0].PASSED,SHIFTHISTORY[1].PASSED,1) COP(SHIFTHISTORY[0].FAILED,SHIFTHISTORY[1].FAILED,1) COP(SHIFTHISTORY[0].EFFICIENT,SHIFTHISTORY[1].EFFICIENT,1) ,COP(CURRENT_SHIFT.COMPLETED,SHIFTHISTORY[0].COMPLETED,1) COP(CURRENT_SHIFT.PASSED,SHIFTHISTORY[0].PASSED,1) COP(CURRENT_SHIFT.FAILED,SHIFTHISTORY[0].FAILED,1) COP(CURRENT_SHIFT.EFFICIENT,SHIFTHISTORY[0].EFFICIENT,1) ]OTE(RESET_STATS);
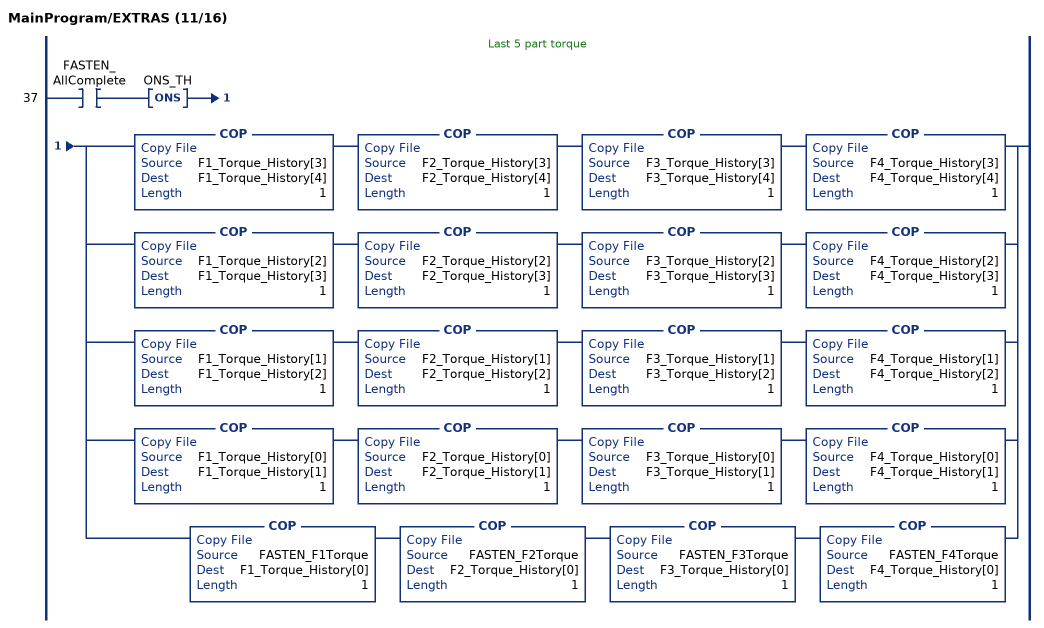
   // Last 5 part torque
   37: XIC(FASTEN_AllComplete)ONS(ONS_TH)[COP(F1_Torque_History[3],F1_Torque_History[4],1) COP(F2_Torque_History[3],F2_Torque_History[4],1) COP(F3_Torque_History[3],F3_Torque_History[4],1) COP(F4_Torque_History[3],F4_Torque_History[4],1) ,COP(F1_Torque_History[2],F1_Torque_History[3],1) COP(F2_Torque_History[2],F2_Torque_History[3],1) COP(F3_Torque_History[2],F3_Torque_History[3],1) COP(F4_Torque_History[2],F4_Torque_History[3],1) ,COP(F1_Torque_History[1],F1_Torque_History[2],1) COP(F2_Torque_History[1],F2_Torque_History[2],1) COP(F3_Torque_History[1],F3_Torque_History[2],1) COP(F4_Torque_History[1],F4_Torque_History[2],1) ,COP(F1_Torque_History[0],F1_Torque_History[1],1) COP(F2_Torque_History[0],F2_Torque_History[1],1) COP(F3_Torque_History[0],F3_Torque_History[1],1) COP(F4_Torque_History[0],F4_Torque_History[1],1) ,COP(FASTEN_F1Torque,F1_Torque_History[0],1) COP(FASTEN_F2Torque,F2_Torque_History[0],1) COP(FASTEN_F3Torque,F3_Torque_History[0],1) COP(FASTEN_F4Torque,F4_Torque_History[0],1) ];
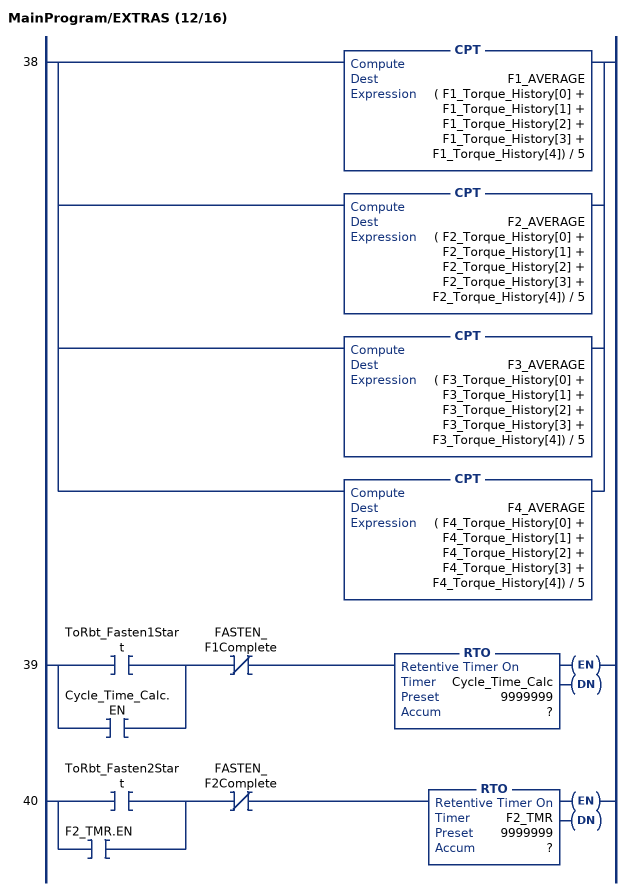
   38: [CPT(F1_AVERAGE,( F1_Torque_History[0] + F1_Torque_History[1] + F1_Torque_History[2] + F1_Torque_History[3] + F1_Torque_History[4]) / 5) ,CPT(F2_AVERAGE,( F2_Torque_History[0] + F2_Torque_History[1] + F2_Torque_History[2] + F2_Torque_History[3] + F2_Torque_History[4]) / 5) ,CPT(F3_AVERAGE,( F3_Torque_History[0] + F3_Torque_History[1] + F3_Torque_History[2] + F3_Torque_History[3] + F3_Torque_History[4]) / 5) ,CPT(F4_AVERAGE,( F4_Torque_History[0] + F4_Torque_History[1] + F4_Torque_History[2] + F4_Torque_History[3] + F4_Torque_History[4]) / 5) ];
   39: [XIC(ToRbt_Fasten1Start) ,XIC(Cycle_Time_Calc.EN) ]XIO(FASTEN_F1Complete)RTO(Cycle_Time_Calc,?,?);
   40: [XIC(ToRbt_Fasten2Start) ,XIC(F2_TMR.EN) ]XIO(FASTEN_F2Complete)RTO(F2_TMR,?,?);
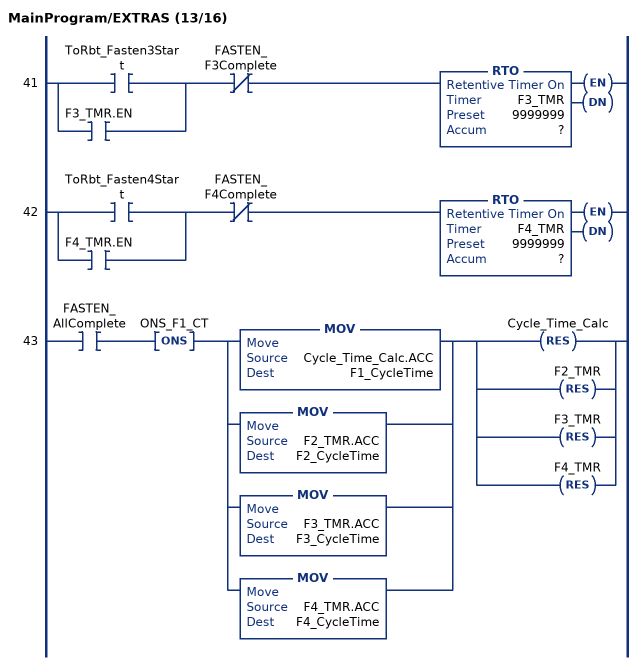
   41: [XIC(ToRbt_Fasten3Start) ,XIC(F3_TMR.EN) ]XIO(FASTEN_F3Complete)RTO(F3_TMR,?,?);
   42: [XIC(ToRbt_Fasten4Start) ,XIC(F4_TMR.EN) ]XIO(FASTEN_F4Complete)RTO(F4_TMR,?,?);
   43: XIC(FASTEN_AllComplete)ONS(ONS_F1_CT)[MOV(Cycle_Time_Calc.ACC,F1_CycleTime) ,MOV(F2_TMR.ACC,F2_CycleTime) ,MOV(F3_TMR.ACC,F3_CycleTime) ,MOV(F4_TMR.ACC,F4_CycleTime) ][RES(Cycle_Time_Calc) ,RES(F2_TMR) ,RES(F3_TMR) ,RES(F4_TMR) ];
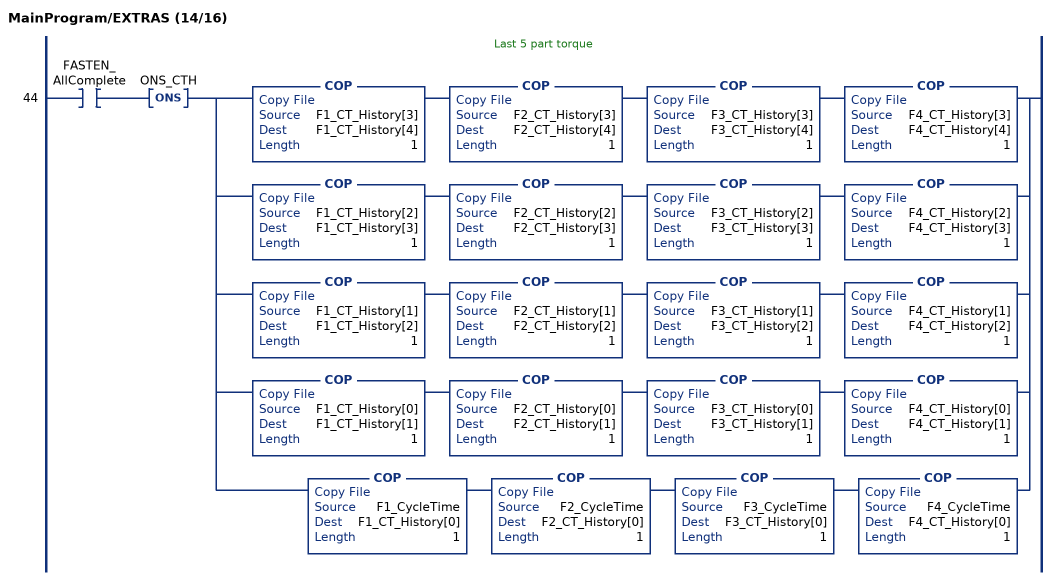
   // Last 5 part torque
   44: XIC(FASTEN_AllComplete)ONS(ONS_CTH)[COP(F1_CT_History[3],F1_CT_History[4],1) COP(F2_CT_History[3],F2_CT_History[4],1) COP(F3_CT_History[3],F3_CT_History[4],1) COP(F4_CT_History[3],F4_CT_History[4],1) ,COP(F1_CT_History[2],F1_CT_History[3],1) COP(F2_CT_History[2],F2_CT_History[3],1) COP(F3_CT_History[2],F3_CT_History[3],1) COP(F4_CT_History[2],F4_CT_History[3],1) ,COP(F1_CT_History[1],F1_CT_History[2],1) COP(F2_CT_History[1],F2_CT_History[2],1) COP(F3_CT_History[1],F3_CT_History[2],1) COP(F4_CT_History[1],F4_CT_History[2],1) ,COP(F1_CT_History[0],F1_CT_History[1],1) COP(F2_CT_History[0],F2_CT_History[1],1) COP(F3_CT_History[0],F3_CT_History[1],1) COP(F4_CT_History[0],F4_CT_History[1],1) ,COP(F1_CycleTime,F1_CT_History[0],1) COP(F2_CycleTime,F2_CT_History[0],1) COP(F3_CycleTime,F3_CT_History[0],1) COP(F4_CycleTime,F4_CT_History[0],1) ];
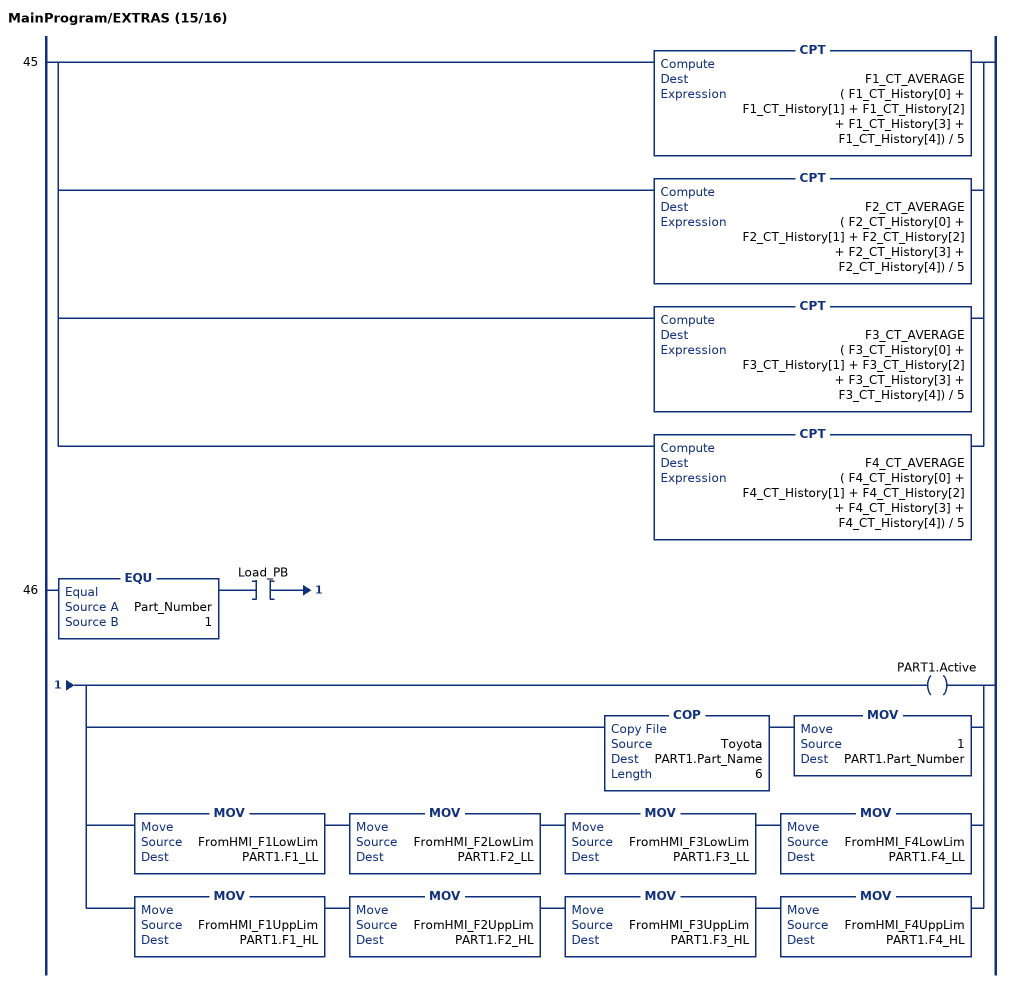
   45: [CPT(F1_CT_AVERAGE,( F1_CT_History[0] + F1_CT_History[1] + F1_CT_History[2] + F1_CT_History[3] + F1_CT_History[4]) / 5) ,CPT(F2_CT_AVERAGE,( F2_CT_History[0] + F2_CT_History[1] + F2_CT_History[2] + F2_CT_History[3] + F2_CT_History[4]) / 5) ,CPT(F3_CT_AVERAGE,( F3_CT_History[0] + F3_CT_History[1] + F3_CT_History[2] + F3_CT_History[3] + F3_CT_History[4]) / 5) ,CPT(F4_CT_AVERAGE,( F4_CT_History[0] + F4_CT_History[1] + F4_CT_History[2] + F4_CT_History[3] + F4_CT_History[4]) / 5) ];
   46: EQU(Part_Number,1)XIC(Load_PB)[OTE(PART1.Active) ,COP(Toyota,PART1.Part_Name,6) MOV(1,PART1.Part_Number) ,MOV(FromHMI_F1LowLim,PART1.F1_LL) MOV(FromHMI_F2LowLim,PART1.F2_LL) MOV(FromHMI_F3LowLim,PART1.F3_LL) MOV(FromHMI_F4LowLim,PART1.F4_LL) ,MOV(FromHMI_F1UppLim,PART1.F1_HL) MOV(FromHMI_F2UppLim,PART1.F2_HL) MOV(FromHMI_F3UppLim,PART1.F3_HL) MOV(FromHMI_F4UppLim,PART1.F4_HL) ];
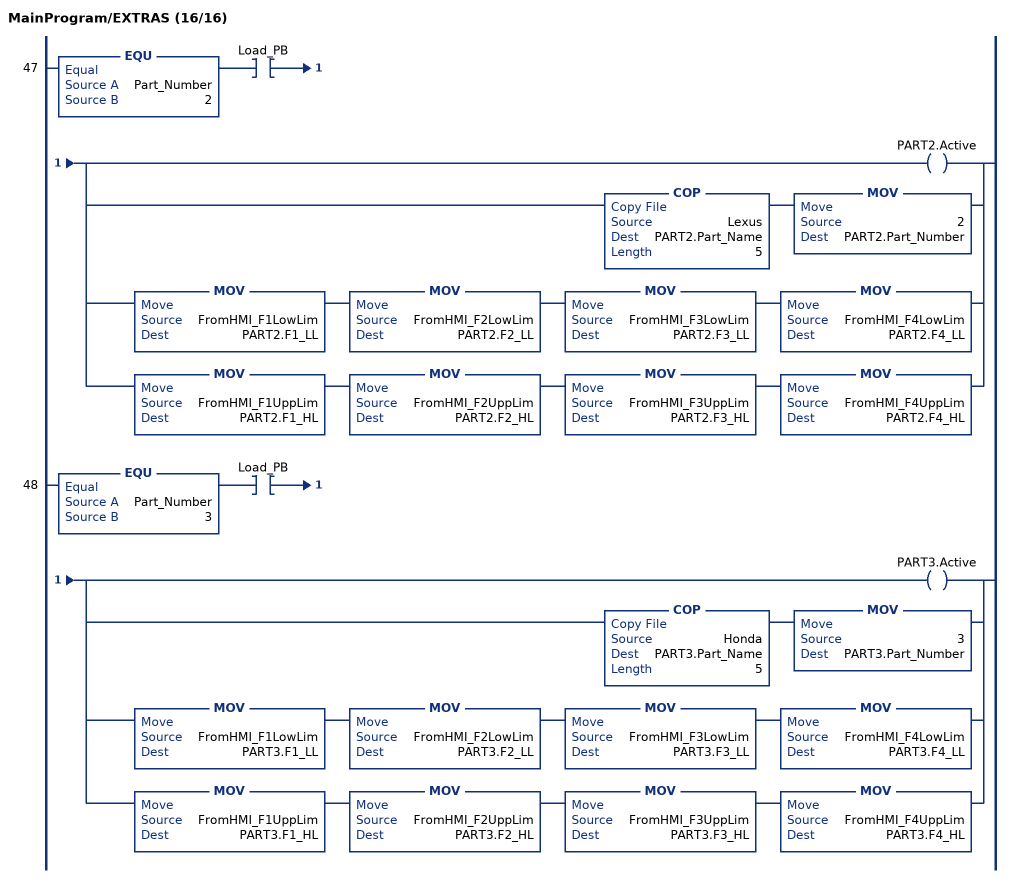
   47: EQU(Part_Number,2)XIC(Load_PB)[OTE(PART2.Active) ,COP(Lexus,PART2.Part_Name,5) MOV(2,PART2.Part_Number) ,MOV(FromHMI_F1LowLim,PART2.F1_LL) MOV(FromHMI_F2LowLim,PART2.F2_LL) MOV(FromHMI_F3LowLim,PART2.F3_LL) MOV(FromHMI_F4LowLim,PART2.F4_LL) ,MOV(FromHMI_F1UppLim,PART2.F1_HL) MOV(FromHMI_F2UppLim,PART2.F2_HL) MOV(FromHMI_F3UppLim,PART2.F3_HL) MOV(FromHMI_F4UppLim,PART2.F4_HL) ];
   48: EQU(Part_Number,3)XIC(Load_PB)[OTE(PART3.Active) ,COP(Honda,PART3.Part_Name,5) MOV(3,PART3.Part_Number) ,MOV(FromHMI_F1LowLim,PART3.F1_LL) MOV(FromHMI_F2LowLim,PART3.F2_LL) MOV(FromHMI_F3LowLim,PART3.F3_LL) MOV(FromHMI_F4LowLim,PART3.F4_LL) ,MOV(FromHMI_F1UppLim,PART3.F1_HL) MOV(FromHMI_F2UppLim,PART3.F2_HL) MOV(FromHMI_F3UppLim,PART3.F3_HL) MOV(FromHMI_F4UppLim,PART3.F4_HL) ];
END_ROUTINE
